FUNCTION_BLOCK SUBLLP8 (* Eight-variable logic proxy to local Subscriber with interface of the globl one *)
  (* Standard: 61499-2 *)
  (* Version 0.0, 2000-11-27, JHC, Rockwell Automation, Saved for CODEC_TEST *)
  (* Compiler header: package fb.rt.vnet;import fb.rt.net.*; *)
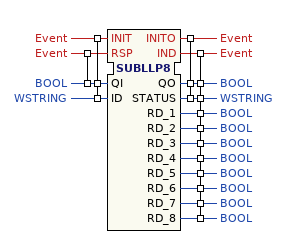
  EVENT_INPUT
    INIT WITH QI, ID; (* Service Initialization *)
    RSP WITH QI; (* Service Response *)
  END_EVENT
  EVENT_OUTPUT
    INITO WITH QO, STATUS; (* Initialization Confirm *)
    IND WITH QO, STATUS, RD_1, RD_2, RD_3, RD_4, RD_5, RD_6, RD_7, RD_8; (* Service Indication *)
  END_EVENT
  VAR_INPUT
    QI : BOOL; (* Event Input Qualifier *)
    ID : WSTRING; (* Connection Identifier *)
  END_VAR
  VAR_OUTPUT
    QO : BOOL; (* Event Output Qualifier *)
    STATUS : WSTRING; (* Service Status *)
    RD_1 : BOOL; (* Subscribed Data *)
    RD_2 : BOOL; (* Subscribed Data *)
    RD_3 : BOOL; (* Subscribed Data *)
    RD_4 : BOOL; (* Subscribed Data *)
    RD_5 : BOOL; (* Subscribed Data *)
    RD_6 : BOOL; (* Subscribed Data *)
    RD_7 : BOOL; (* Subscribed Data *)
    RD_8 : BOOL; (* Subscribed Data *)
  END_VAR
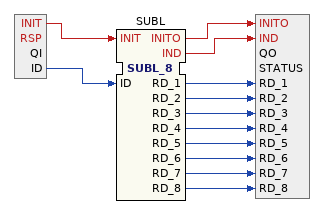
  FBS
    SUBL : SUBL_8;
  END_FBS
  EVENT_CONNECTIONS
    INIT TO SUBL.INIT;
    SUBL.INITO TO INITO;
    SUBL.IND TO IND;
  END_CONNECTIONS
  DATA_CONNECTIONS
    ID TO SUBL.ID;
    SUBL.RD_1 TO RD_1;
    SUBL.RD_2 TO RD_2;
    SUBL.RD_3 TO RD_3;
    SUBL.RD_4 TO RD_4;
    SUBL.RD_5 TO RD_5;
    SUBL.RD_6 TO RD_6;
    SUBL.RD_7 TO RD_7;
    SUBL.RD_8 TO RD_8;
  END_CONNECTIONS
END_FUNCTION_BLOCK
